{attribute 'GeneratedUsingTerminal: EL6021-0000-0018'}
{attribute addProperty BoxType "EL6021-0000-0018"}
{attribute addProperty Id "CtrlAT %Q*Ctrl_71604E865Data_OutAT %Q*ARRAY[0..21] OF USINT22"}
{attribute addProperty CRC "2695605661"}
{attribute addProperty Size "27"}
TYPE COM_RxPDO_Map_Outputs_DEF408EC EXTENDS OutputBase_10CEE7DE :
STRUCT
	{attribute addProperty Name "Ctrl"}
	Ctrl AT %Q* : Ctrl_71604E86;
	{attribute addProperty Name "Data_Out"}
	Data_Out AT %Q* : ARRAY[0..21] OF USINT;
END_STRUCT
END_TYPE

(* stored: Version 1.2.0.0, ProductVersion 3.1.4024.11
   DUT COM_RxPDO_Map_Outputs_DEF408EC: Id {f746064b-014a-4a6a-932d-f329a09e7f08} *)
